FUNCTION_BLOCK Mixing
VAR_INPUT
	diEnabled : BOOL;
	iSecImp : BOOL;
END_VAR
VAR_OUTPUT
	doEnabled : BOOL;
END_VAR
VAR_IN_OUT
	MixingPhase : TPhaseMixing;
	MixerEng : TEngine;
END_VAR
VAR
END_VAR

{region "Aut/Man"}
    // switching state of engine - automatic or manual control (default state is manual)
  
{endregion}

{region "ManCtrl"}
    // processing manual actions - if command is processed, it is sets to FALSE even if can't be processed
    // Phase commands are start, stop, pause and resume 
    // Start - start mixing  
    // Stop - stop mixing
    // Pause - stop mixing 
    // Resume - start mixing
    // real states of phase are writed into states in phase structure
   
{endregion}

{region "AutCtrl"}
    // if request to run in automatic mode -> set auto request to mixing to 1, if not request to mixing is 0
    // commands should be sets to false after their processing
   
{endregion}

{region "Done"}
    // every phase should have finish condition - mixing phase - if time of runnig is bigger or same as requested
    // after that done state should be setted to 1
 
{endregion}

{region "States"}
    //Command mixer in cases of states

{endregion}


// delault state of phase - if not any state sets state to idle
IF NOT MixingPhase.State.Idle AND NOT MixingPhase.State.Done AND NOT MixingPhase.State.Paused AND NOT MixingPhase.State.Running THEN
    MixingPhase.State.Idle := 1;
END_IF;


// delault state of phase - if not any state sets state to idle
IF MixingPhase.State.Idle THEN
    MixingPhase.State.StateInt := Global.PhIdle;
ELSIF MixingPhase.State.Running THEN
    MixingPhase.State.StateInt := Global.PhRunning;
ELSE
    MixingPhase.State.StateInt := Global.PhPause;
END_IF;

doEnabled := diEnabled;

END_FUNCTION_BLOCK

(* stored: Version 1.1.0.1, ProductVersion 3.1.4024.13
   POU Mixing: Id {c7d77201-326e-43f5-84be-5e5d3f37b70d}, SpecialFunc None *)
